// TIA Portal V19 export
TYPE "LAF_typeChecksum"
TITLE = Structure PLC checksum / Strukrur PLC Checksum
// Type contains all information which is shown in the visualization. / PLC Checksum
// stored: Access Published
   STRUCT
      checksumStandard { ExternalWritable := 'False'} : String[16];   // Checksumme Standard Bausteine / Checksum standard blocks
      checksumStandardOld { ExternalWritable := 'False'} : String[16];   // Checksumme Standard Bausteine (Alt) / Checksum standard blocks (Old)
      checksumSafety { ExternalWritable := 'False'} : String[16];   // Checksumme Safety Bausteine / Checksum safety blocks
      checksumSafetyOld { ExternalWritable := 'False'} : String[16];   // Checksumme Safety Bausteine (Alt) / Checksum safety blocks (Old)
      checksumTextlists { ExternalWritable := 'False'} : String[16];   // Checksumme Textlisten / Checksum text lists
      checksumTextlistsOld { ExternalWritable := 'False'} : String[16];   // Checksumme Textlisten (Alt) / Checksum text lists (Old)
      dateTimeStandardModified { ExternalWritable := 'False'} : Date_And_Time;   // Standard Bausteine modifiziert Datum&Uhrzeit / Standard blocks modified Date&Time
      dateTimeSafetyModified { ExternalWritable := 'False'} : Date_And_Time;   // Safety Bausteine modifiziert Datum&Uhrzeit / Safety blocks modified Date&Time
      dateTimeTextlistModified { ExternalWritable := 'False'} : Date_And_Time;   // Textlisten modifiziert Datum&Uhrzeit / Textlists modified Date&Time
      standardModified { ExternalWritable := 'False'} : Bool;   // Standard Bausteine wurden geändert / Standard blocks are modified
      safetyModified { ExternalWritable := 'False'} : Bool;   // Safety Bausteine wurden geändert / Safety blocks are modified
      textlistsModified { ExternalWritable := 'False'} : Bool;   // Textlisten wurden geändert / Textlists are modified
      summaryModified { ExternalWritable := 'False'} : Bool;   // Summensignal Änderung / Summary modified
      updateValuesOld : Bool;   // Aktualisiere Altwerte / Update old values
   END_STRUCT;
END_TYPE
